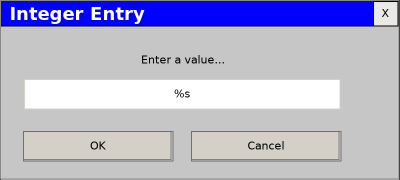
VISUALIZATION dialogEnterValueInteger  // 400x180
VAR_IN_OUT
	enteredValue:INT;
END_VAR
    Rectangle (0,0 400x188)
    Rectangle (0,0 400x26), "Integer Entry"
    Rectangle (373,1 25x25), "X"
        OnMouseClick: CloseDialog Dialog=dialogEnterValueInteger, Result=Cancel, NumpadKeypadSet=True
    Label (108,45 150x30), "Enter a value..."
    Textfield (24,79 316x30), "%s", text variable: enteredValue
        OnMouseClick: write enteredValue via VisuDialogs.Numpad
    Button (23,131 150x30), "OK"
        OnMouseClick: CloseDialog Dialog=dialogEnterValueInteger, Result=OK, NumpadKeypadSet=True
    Button (191,131 150x30), "Cancel"
        OnMouseClick: CloseDialog Dialog=dialogEnterValueInteger, Result=Cancel, NumpadKeypadSet=True
END_VISUALIZATION

(* stored: Version 1.1.0.1, ProductVersion 3.1.4024.11
   Visu dialogEnterValueInteger: Id {b76d4f99-cc78-0d37-0858-189febf7fb16} *)
